// TIA Portal V20 export
DATA_BLOCK "TestTempDB"   // DB502
// stored: MemoryReserve 100
   VAR
      TempBool : Array[0..100] of Bool;
   END_VAR
BEGIN
END_DATA_BLOCK
